FUNCTION_BLOCK LocalCylinderControl (* Basic Function Block Type *)
  (* Standard: 61499-2 *)
  (* Version 0.0, 12/9/2021, e_net, nxtControl GmbH, Template *)
  PACKAGE Main;
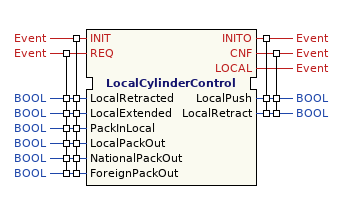
  EVENT_INPUT
    INIT WITH LocalRetracted, LocalExtended, PackInLocal, LocalPackOut, NationalPackOut, ForeignPackOut; (* Initialization Request *)
    REQ WITH LocalRetracted, LocalExtended, PackInLocal, LocalPackOut, NationalPackOut, ForeignPackOut; (* Normal Execution Request *)
  END_EVENT
  EVENT_OUTPUT
    INITO WITH LocalPush, LocalRetract; (* Initialization Confirm *)
    CNF WITH LocalPush, LocalRetract; (* Execution Confirmation *)
    LOCAL;
  END_EVENT
  VAR_INPUT
    LocalRetracted : BOOL; (* Input event qualifier *)
    LocalExtended : BOOL;
    PackInLocal : BOOL;
    LocalPackOut : BOOL;
    NationalPackOut : BOOL;
    ForeignPackOut : BOOL;
  END_VAR
  VAR_OUTPUT
    LocalPush : BOOL; (* Output event qualifier *)
    LocalRetract : BOOL;
  END_VAR
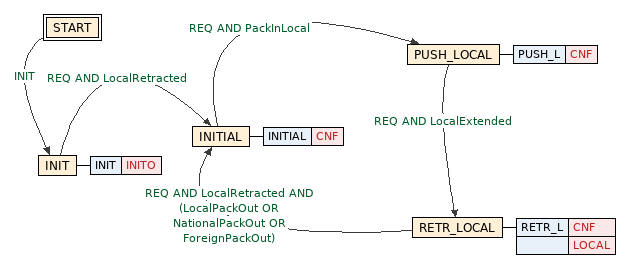
  EC_STATES
    START; (* Initial State *)
    INIT : INIT -> INITO; (* Initialization *)
    INITIAL : INITIAL -> CNF;
    PUSH_LOCAL : PUSH_L -> CNF;
    RETR_LOCAL : RETR_L -> CNF, -> LOCAL;
  END_STATES
  EC_TRANSITIONS
    START TO INIT := INIT;
    INIT TO INITIAL := REQ AND LocalRetracted;
    INITIAL TO PUSH_LOCAL := REQ AND PackInLocal;
    RETR_LOCAL TO INITIAL := REQ AND LocalRetracted AND (LocalPackOut OR NationalPackOut OR ForeignPackOut);
    PUSH_LOCAL TO RETR_LOCAL := REQ AND LocalExtended;
  END_TRANSITIONS
  ALGORITHM INIT IN ST: (* Initialization algorithm *)
LocalPush:= FALSE;
LocalRetract:= TRUE;
  END_ALGORITHM
  ALGORITHM INITIAL IN ST:
LocalRetract:=FALSE;
  END_ALGORITHM
  ALGORITHM PUSH_L IN ST:
LocalPush:=TRUE;
  END_ALGORITHM
  ALGORITHM RETR_L IN ST:
LocalPush:=FALSE;
LocalRetract:=TRUE;
  END_ALGORITHM
END_FUNCTION_BLOCK
